{attribute 'pack_mode' := '2'}
TYPE ST_MOVER_STATE :
STRUCT
  State           : E_MOVER_STATE;  // ST_MOVER_CTRL.Cmd with added E_PROGRESS
  MasterId        : USINT;            // mirror NC AxisId of Master axis
END_STRUCT
END_TYPE

(* stored: Version 1.1.0.1
   DUT ST_MOVER_STATE: Id {c9ad9fb0-b875-49f0-bd31-39da0e79c978} *)
